Staubli VAL3: onF6Event.pgx

program onF6Event(bool& x_bSave[] (dimensions=1))
begin
  // look if the bButton is enable
  if bButton[5] and saveData:mode>1
    //
    // CHANGE PLC STATUS
    //
    if saveData:bPlc
      cycleStatus:nInterfaceToSV=11
    else
      cycleStatus:nInterfaceToSV=10
    endIf
    wait(cycleStatus:nInterfaceToSV==-1)
    logMsg("[KERNEL] INTERFACE:Change PLC STATUS")
    x_bSave=true
  endIf
end
